// TIA Portal V17 export
// export: Created 2022-04-06T07:28:37.7441139Z, ExportSetting WithDefaults, DisplayName Totally Integrated Automation Portal, DisplayVersion V17, DisplayName TIA Portal Openness, DisplayVersion V17, DisplayName TIA Portal Version Control Interface, DisplayVersion V17, DisplayName TIA Portal Test Suite Advanced, DisplayVersion V17, DisplayName SINAMICS Startdrive Advanced, DisplayVersion V17, DisplayName SINAMICS Startdrive G130, G150, S120, S150, SINAMICS MV, S210, DisplayVersion V17, DisplayName SINAMICS Startdrive G110M, G120, G120C, G120D, G120P, G115D, DisplayVersion V17, DisplayName STEP 7 Professional, DisplayVersion V17, DisplayName STEP 7 Safety, DisplayVersion V17, DisplayName WinCC Advanced / Unified PC, DisplayVersion V17
ORGANIZATION_BLOCK "Main"   // OB1, LAD, ProgramCycle
TITLE = "Main Program Sweep (Cycle)"
{ S7_Optimized_Access := 'TRUE' }
VERSION : 0.1
// stored: AutoNumber true, IsIECCheckEnabled false, SetENOAutomatically false
   VAR_INPUT
      Initial_Call : Bool;   // Initial call of this OB
      Remanence : Bool;   // =True, if remanent data are available
   END_VAR
BEGIN

REGION Network 2
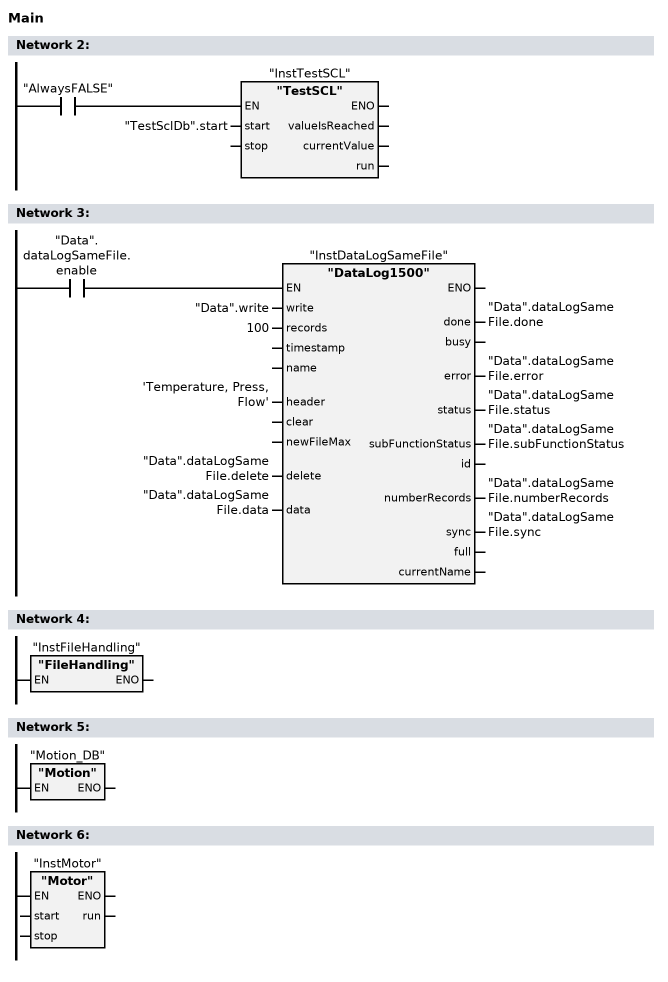
   RUNG wire#powerrail
      Contact( "AlwaysFALSE" )
      "InstTestSCL"(start := "TestSclDb".start, valueIsReached =>, currentValue =>, stop :=, run =>)
   END_RUNG
   // the same network as SCL:
   IF "AlwaysFALSE" THEN
       "InstTestSCL"(start := "TestSclDb".start);   // "TestSCL"
   END_IF;
END_REGION

REGION Network 3
   RUNG wire#powerrail
      Contact( "Data".dataLogSameFile.enable )
      "InstDataLogSameFile"(write := "Data".write, records := 100, timestamp :=, "name" :=, header := 'Temperature, Press, Flow', clear :=, newFileMax :=, delete := "Data".dataLogSameFile.delete, data := "Data".dataLogSameFile.data, done => "Data".dataLogSameFile.done, busy =>, error => "Data".dataLogSameFile.error, status => "Data".dataLogSameFile.status, subFunctionStatus => "Data".dataLogSameFile.subFunctionStatus, id =>, numberRecords => "Data".dataLogSameFile.numberRecords, sync => "Data".dataLogSameFile.sync, full =>, currentName =>)
   END_RUNG
   // the same network as SCL:
   IF "Data".dataLogSameFile.enable THEN
       "InstDataLogSameFile"(write := "Data".write,   // "DataLog1500"
                             records := 100,
                             header := 'Temperature, Press, Flow',
                             delete := "Data".dataLogSameFile.delete,
                             data := "Data".dataLogSameFile.data,
                             done => "Data".dataLogSameFile.done,
                             error => "Data".dataLogSameFile.error,
                             status => "Data".dataLogSameFile.status,
                             subFunctionStatus => "Data".dataLogSameFile.subFunctionStatus,
                             numberRecords => "Data".dataLogSameFile.numberRecords,
                             sync => "Data".dataLogSameFile.sync);
   END_IF;
END_REGION

REGION Network 4
   RUNG wire#powerrail
      "InstFileHandling"()
   END_RUNG
   // the same network as SCL:
   "InstFileHandling"();   // "FileHandling"
END_REGION

REGION Network 5
   RUNG wire#powerrail
      "Motion_DB"()
   END_RUNG
   // the same network as SCL:
   "Motion_DB"();   // "Motion"
END_REGION

REGION Network 6
   RUNG wire#powerrail
      "InstMotor"(start :=, stop :=, run =>)
   END_RUNG
   // the same network as SCL:
   "InstMotor"();   // "Motor"
END_REGION
END_ORGANIZATION_BLOCK
